FUNCTION_BLOCK FB_Manual_PC
VAR_INPUT
	bEnable					: BOOL;
END_VAR
VAR_OUTPUT
	fPCV					: LREAL;
	fSCV					: LREAL;
END_VAR
VAR
	//Function Blocks
	fbJoystick				: FB_Joystick;
	fbGetStartPos			: FB_StartPos;
	fbWinchVelIntegrator	: FB_Integrator;
	fbPID_Controller		: FB_PID_Controller;
	fbMUX_selector			: FB_MUX_selector;
	
	//Manual PosRef
	fWinchVelRefManual		: LREAL;
	fWInchVelRefAuto		: LREAL; //Brukes ikke
	fInitialWinchPos		: LREAL;
	
	//Valve signals
	fPCV_Manual			: LREAL;
	fPCV_PosRef			: LREAL;
	fPCV_Off			: LREAL;
	fSCV_On				: LREAL;
	fSCV_Off			: LREAL;
	
	
	//Notat på hva som skal til OPC UA
	//G_Motion_Control.fWinchPosRefManual
	


	END_VAR
VAR // added by the converter: edge detectors and wires of the graphical bodies
    _w1 : BOOL;
END_VAR

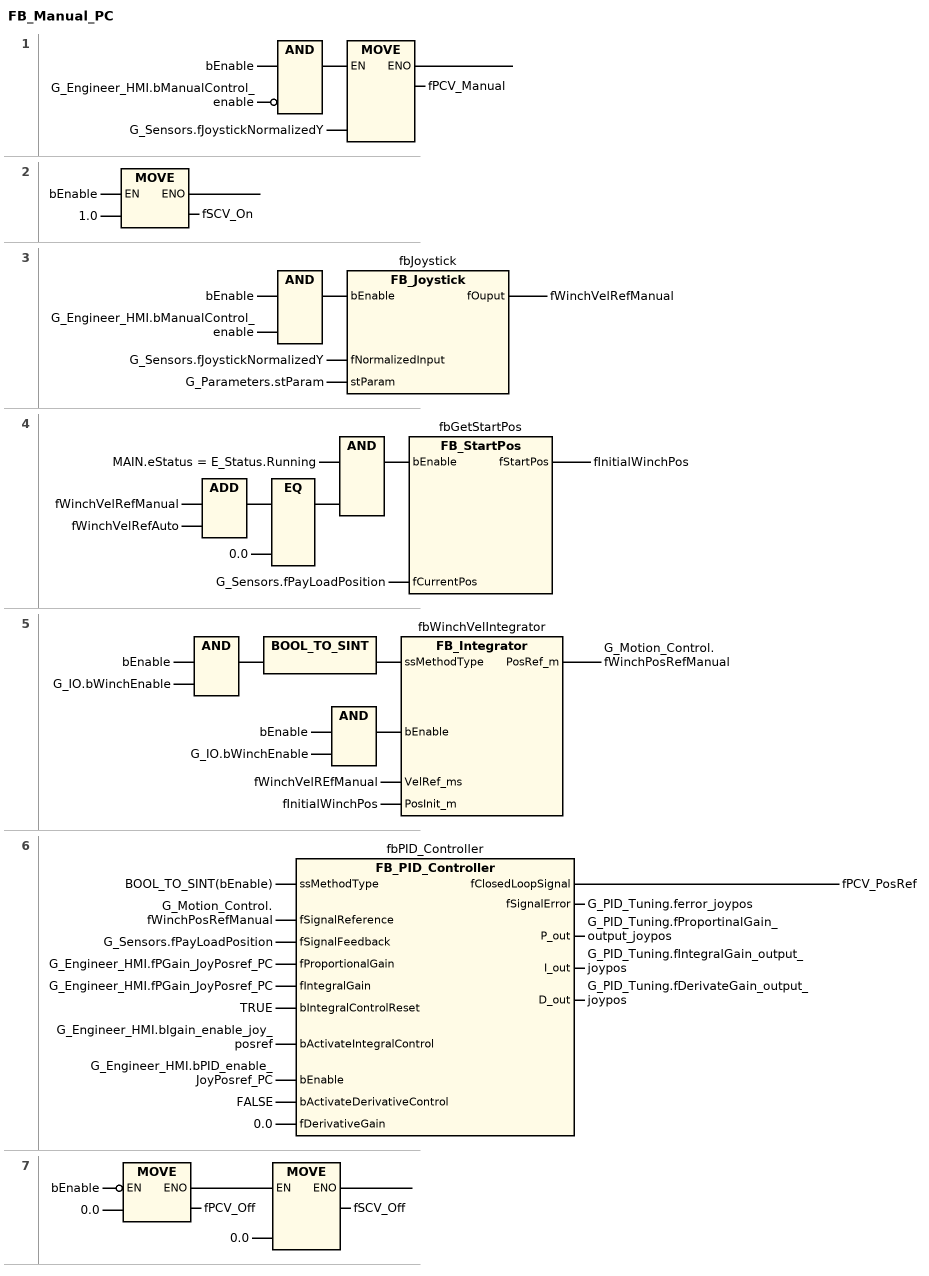
// NETWORK 1
IF bEnable AND NOT G_Engineer_HMI.bManualControl_enable THEN fPCV_Manual := G_Sensors.fJoystickNormalizedY; END_IF

// NETWORK 2
IF bEnable THEN fSCV_On := 1.0; END_IF

// NETWORK 3
fbJoystick(
    bEnable := bEnable AND G_Engineer_HMI.bManualControl_enable,
    fNormalizedInput := G_Sensors.fJoystickNormalizedY,
    stParam := G_Parameters.stParam); // FB_Joystick
fWinchVelRefManual := fbJoystick.fOuput;

// NETWORK 4
fbGetStartPos(bEnable := (MAIN.eStatus = E_Status.Running) AND fWinchVelRefManual + fWinchVelRefAuto = 0.0, fCurrentPos := G_Sensors.fPayLoadPosition); // FB_StartPos
fInitialWinchPos := fbGetStartPos.fStartPos;

// NETWORK 5
fbWinchVelIntegrator(
    ssMethodType := BOOL_TO_SINT(bEnable AND G_IO.bWinchEnable),
    bEnable := bEnable AND G_IO.bWinchEnable,
    VelRef_ms := fWinchVelREfManual,
    PosInit_m := fInitialWinchPos); // FB_Integrator
G_Motion_Control.fWinchPosRefManual := fbWinchVelIntegrator.PosRef_m;

// NETWORK 6
fbPID_Controller(
    ssMethodType := BOOL_TO_SINT(bEnable),
    fSignalReference := G_Motion_Control.fWinchPosRefManual,
    fSignalFeedback := G_Sensors.fPayLoadPosition,
    fProportionalGain := G_Engineer_HMI.fPGain_JoyPosref_PC,
    fIntegralGain := G_Engineer_HMI.fPGain_JoyPosref_PC,
    bIntegralControlReset := TRUE,
    bActivateIntegralControl := G_Engineer_HMI.bIgain_enable_joy_posref,
    bEnable := G_Engineer_HMI.bPID_enable_JoyPosref_PC,
    bActivateDerivativeControl := FALSE,
    fDerivativeGain := 0.0,
    fSignalError => G_PID_Tuning.ferror_joypos,
    P_out => G_PID_Tuning.fProportinalGain_output_joypos,
    I_out => G_PID_Tuning.fIntegralGain_output_joypos,
    D_out => G_PID_Tuning.fDerivateGain_output_joypos); // FB_PID_Controller
fPCV_PosRef := fbPID_Controller.fClosedLoopSignal;

// NETWORK 7
_w1 := NOT bEnable;
IF _w1 THEN fPCV_Off := 0.0; END_IF
IF _w1 THEN fSCV_Off := 0.0; END_IF

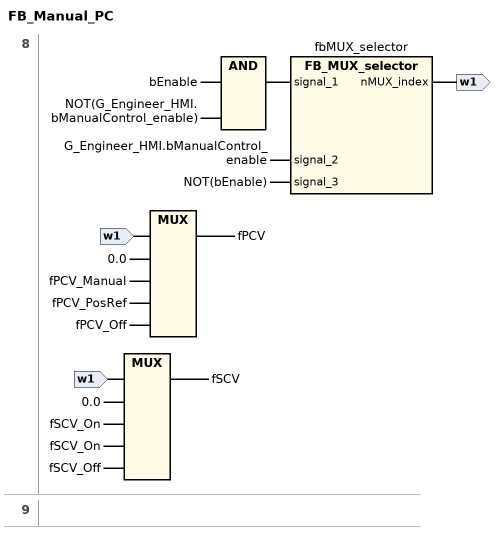
// NETWORK 8
fbMUX_selector(
    signal_1 := bEnable AND (NOT(G_Engineer_HMI.bManualControl_enable)),
    signal_2 := G_Engineer_HMI.bManualControl_enable,
    signal_3 := NOT(bEnable)); // FB_MUX_selector
fPCV := MUX(fbMUX_selector.nMUX_index, 0.0, fPCV_Manual, fPCV_PosRef, fPCV_Off);
fSCV := MUX(fbMUX_selector.nMUX_index, 0.0, fSCV_On, fSCV_On, fSCV_Off);

// NETWORK 9

END_FUNCTION_BLOCK

(* stored: Version 1.1.0.1
   POU FB_Manual_PC: Id {ca6322d9-312c-4f2c-9084-e6c81a15149c}, SpecialFunc None *)
